{attribute 'GeneratedUsingTerminal: CU1124-0000-0016'}
{attribute addProperty BoxType "CU1124-0000-0016"}
{attribute addProperty Id "EtcSlaveTerminalBaseInfoDataAT %I*InfoData_6F19DB2B2"}
{attribute addProperty CRC "2874840167"}
{attribute addProperty Size "2"}
TYPE CU1124_AB5A9467 EXTENDS EtcSlaveTerminalBase :
STRUCT
	{attribute addProperty Name "InfoData"}
	InfoData : InfoData_6F19DB2B;
END_STRUCT
END_TYPE

(* stored: Version 1.2.0.0, ProductVersion 3.1.4024.9
   DUT CU1124_AB5A9467: Id {301d093d-f8c3-4155-9cd8-dc7e0cf6c309} *)
